	(* Titlezeile zeichnen *)
	FB_TN_SC_FILL(	Iin_X1 := INT#00,
					Iin_Y1 := INT#00,
					Iin_X2 := INT#79,
					Iin_Y2 := INT#00,
					Iby_CHAR := BYTE#32,
					Iby_Attr := BYTE#16#07,
					Xus_TN_SCREEN := Xus_TN_SCREEN);

	(* Fusszeile zeichnen *)
	FB_TN_SC_FILL(	Iin_X1 := INT#00,
					Iin_Y1 := INT#23,
					Iin_X2 := INT#79,
					Iin_Y2 := INT#23,
					Iby_CHAR := BYTE#32,
					Iby_Attr := BYTE#16#37,
					Xus_TN_SCREEN := Xus_TN_SCREEN);

	(* Rahmen für Viewport zeichnen *)
	FB_TN_SC_BOX(	Iin_X1 := INT#00,
					Iin_Y1 := INT#01,
					Iin_X2 := INT#77,
					Iin_Y2 := INT#17,
					Iby_FILL := BYTE#16#00, (* keine Füllung *)
					Iin_BORDER := INT#02, (* Double-Line Border *)
					Iby_ATTR := BYTE#16#74, (* Weiss , Blau *)
					Xus_TN_SCREEN := Xus_TN_SCREEN);

	(* Shadow für Rahmen von Viewport zeichnen *)
	FB_TN_SC_ADD_SHADOW(Iin_X1 := INT#01,
						Iin_Y1 := INT#02,
						Iin_X2 := INT#78,
						Iin_Y2 := INT#18,
						Iin_OPTION := INT#00,
						Xus_TN_SCREEN := Xus_TN_SCREEN);

	(* Trennlinie Viewport_Data und Commandline zeichnen *)
	FB_TN_SC_LINE(	Iin_X1 := INT#00,
					Iin_Y1 := INT#15,
					Iin_X2 := INT#77,
					Iin_Y2 := INT#15,
					Iby_ATTR := BYTE#16#74,
					Iby_BORDER := BYTE#02,
					Xus_TN_SCREEN := Xus_TN_SCREEN);

	(* Title Viewport zeichnen *)
	FB_TN_SC_WRITE(	Iin_X := INT#29,
					Iin_Y := INT#01,
					Iby_ATTR := BYTE#16#74,
					Ist_STRING := '[ SYSTEM-CONSOLE ]',
					Xus_TN_SCREEN := Xus_TN_SCREEN);

	(* Rahmen für Parameter-Feld zeichnen *)
	FB_TN_SC_BOX(	Iin_X1 := INT#02,
					Iin_Y1 := INT#19,
					Iin_X2 := INT#74,
					Iin_Y2 := INT#21,
					Iby_FILL := BYTE#16#20,
					Iin_BORDER := INT#01, (* Double-Line Border *)
					Iby_ATTR := BYTE#16#74, (* Weiss , Blau *)
					Xus_TN_SCREEN := Xus_TN_SCREEN);

	(* Shadow für Rahmen von Parameter-Feld zeichnen *)
	FB_TN_SC_ADD_SHADOW(Iin_X1 := INT#03,
						Iin_Y1 := INT#20,
						Iin_X2 := INT#75,
						Iin_Y2 := INT#22,
						Iin_OPTION := INT#00,
						Xus_TN_SCREEN := Xus_TN_SCREEN);

	(* Alle Input-Controls initialisieren *)

	Xus_TN_INPUT_CONTROL.bo_Enable := FALSE;

	(* Initialisierung der Eingabe-Zeile *)
	Xus_TN_INPUT_CONTROL.usa_TN_INPUT_CONTROL_DATA[1].in_Type := INT#01;
	Xus_TN_INPUT_CONTROL.usa_TN_INPUT_CONTROL_DATA[1].in_Y := INT#16;
	Xus_TN_INPUT_CONTROL.usa_TN_INPUT_CONTROL_DATA[1].in_X := INT#09;
	Xus_TN_INPUT_CONTROL.usa_TN_INPUT_CONTROL_DATA[1].by_Attr_mF := BYTE#16#72; (* Weiss, Grün *)
	Xus_TN_INPUT_CONTROL.usa_TN_INPUT_CONTROL_DATA[1].by_Attr_oF := BYTE#16#74; (* Weiss, Blau *)
	Xus_TN_INPUT_CONTROL.usa_TN_INPUT_CONTROL_DATA[1].in_Cursor_Pos := INT#0;
	Xus_TN_INPUT_CONTROL.usa_TN_INPUT_CONTROL_DATA[1].bo_Input_Only_Num := FALSE;
	Xus_TN_INPUT_CONTROL.usa_TN_INPUT_CONTROL_DATA[1].bo_Input_Hidden := FALSE;
	Xus_TN_INPUT_CONTROL.usa_TN_INPUT_CONTROL_DATA[1].st_Input_Mask := '                                                                    ';
	Xus_TN_INPUT_CONTROL.usa_TN_INPUT_CONTROL_DATA[1].st_Input_Data := Xus_TN_INPUT_CONTROL.usa_TN_INPUT_CONTROL_DATA[1].st_Input_Mask;
	Xus_TN_INPUT_CONTROL.usa_TN_INPUT_CONTROL_DATA[1].st_Input_ToolTip := 'Eingabezeile aktiv       | SCROLL F1/F2/F3/F4 |';
	Xus_TN_INPUT_CONTROL.usa_TN_INPUT_CONTROL_DATA[1].in_Input_Option := INT#02;
	Xus_TN_INPUT_CONTROL.usa_TN_INPUT_CONTROL_DATA[1].in_Title_Y_Offset := INT#00;
	Xus_TN_INPUT_CONTROL.usa_TN_INPUT_CONTROL_DATA[1].in_Title_X_Offset := INT#00;
	Xus_TN_INPUT_CONTROL.usa_TN_INPUT_CONTROL_DATA[1].by_Title_Attr := BYTE#16#34;
	Xus_TN_INPUT_CONTROL.usa_TN_INPUT_CONTROL_DATA[1].st_Title_String := 'Befehl: ';

	(* Initialisierung Selection Text *)
	Xus_TN_INPUT_CONTROL.usa_TN_INPUT_CONTROL_DATA[2].in_Type := INT#03;
	Xus_TN_INPUT_CONTROL.usa_TN_INPUT_CONTROL_DATA[2].in_Y := INT#20;
	Xus_TN_INPUT_CONTROL.usa_TN_INPUT_CONTROL_DATA[2].in_X := INT#18;
	Xus_TN_INPUT_CONTROL.usa_TN_INPUT_CONTROL_DATA[2].by_Attr_mF := BYTE#16#17;
	Xus_TN_INPUT_CONTROL.usa_TN_INPUT_CONTROL_DATA[2].by_Attr_oF := BYTE#16#47;
	Xus_TN_INPUT_CONTROL.usa_TN_INPUT_CONTROL_DATA[2].st_Input_ToolTip := ' aktuellen LOG-Level aendern     | press enter to select |';
	Xus_TN_INPUT_CONTROL.usa_TN_INPUT_CONTROL_DATA[2].in_Input_Option := INT#00;
	Xus_TN_INPUT_CONTROL.usa_TN_INPUT_CONTROL_DATA[2].in_Title_Y_Offset := INT#00;
	Xus_TN_INPUT_CONTROL.usa_TN_INPUT_CONTROL_DATA[2].in_Title_X_Offset := INT#00;
	Xus_TN_INPUT_CONTROL.usa_TN_INPUT_CONTROL_DATA[2].by_Title_Attr := BYTE#16#34;
	Xus_TN_INPUT_CONTROL.usa_TN_INPUT_CONTROL_DATA[2].st_Title_String := ' LOG-Level ';
	Xus_TN_INPUT_CONTROL.usa_TN_INPUT_CONTROL_DATA[2].st_Input_Mask := '  ';
	Xus_TN_INPUT_CONTROL.usa_TN_INPUT_CONTROL_DATA[2].st_Input_Data := '01#02#03#04#05#06#07#08#09#10#11#12#13#14#15';

	(* Initialisierung Selection Text *)
	Xus_TN_INPUT_CONTROL.usa_TN_INPUT_CONTROL_DATA[3].in_Type := INT#02;
	Xus_TN_INPUT_CONTROL.usa_TN_INPUT_CONTROL_DATA[3].in_Y := INT#20;
	Xus_TN_INPUT_CONTROL.usa_TN_INPUT_CONTROL_DATA[3].in_X := INT#37;
	Xus_TN_INPUT_CONTROL.usa_TN_INPUT_CONTROL_DATA[3].by_Attr_mF := BYTE#16#17;
	Xus_TN_INPUT_CONTROL.usa_TN_INPUT_CONTROL_DATA[3].by_Attr_oF := BYTE#16#47;
	Xus_TN_INPUT_CONTROL.usa_TN_INPUT_CONTROL_DATA[3].st_Input_ToolTip := ' Optionline aktiv      | press space to select |';
	Xus_TN_INPUT_CONTROL.usa_TN_INPUT_CONTROL_DATA[3].in_Input_Option := INT#02;
	Xus_TN_INPUT_CONTROL.usa_TN_INPUT_CONTROL_DATA[3].in_Title_Y_Offset := INT#00;
	Xus_TN_INPUT_CONTROL.usa_TN_INPUT_CONTROL_DATA[3].in_Title_X_Offset := INT#00;
	Xus_TN_INPUT_CONTROL.usa_TN_INPUT_CONTROL_DATA[3].by_Title_Attr := BYTE#16#34;
	Xus_TN_INPUT_CONTROL.usa_TN_INPUT_CONTROL_DATA[3].st_Title_String := '  Selektion  ';
	Xus_TN_INPUT_CONTROL.usa_TN_INPUT_CONTROL_DATA[3].st_Input_Mask := '     ';
	Xus_TN_INPUT_CONTROL.usa_TN_INPUT_CONTROL_DATA[3].st_Input_Data := '[ ]#[x]';

	(* Initialisierung Selection Text *)
	Xus_TN_INPUT_CONTROL.usa_TN_INPUT_CONTROL_DATA[4].in_Type := INT#02;
	Xus_TN_INPUT_CONTROL.usa_TN_INPUT_CONTROL_DATA[4].in_Y := INT#20;
	Xus_TN_INPUT_CONTROL.usa_TN_INPUT_CONTROL_DATA[4].in_X := INT#58;
	Xus_TN_INPUT_CONTROL.usa_TN_INPUT_CONTROL_DATA[4].by_Attr_mF := BYTE#16#17;
	Xus_TN_INPUT_CONTROL.usa_TN_INPUT_CONTROL_DATA[4].by_Attr_oF := BYTE#16#47;
	Xus_TN_INPUT_CONTROL.usa_TN_INPUT_CONTROL_DATA[4].st_Input_ToolTip := ' Selektion-Text aktiv      | press space to select |';
	Xus_TN_INPUT_CONTROL.usa_TN_INPUT_CONTROL_DATA[4].in_Input_Option := INT#02;
	Xus_TN_INPUT_CONTROL.usa_TN_INPUT_CONTROL_DATA[4].in_Title_Y_Offset := INT#00;
	Xus_TN_INPUT_CONTROL.usa_TN_INPUT_CONTROL_DATA[4].in_Title_X_Offset := INT#00;
	Xus_TN_INPUT_CONTROL.usa_TN_INPUT_CONTROL_DATA[4].by_Title_Attr := BYTE#16#34;
	Xus_TN_INPUT_CONTROL.usa_TN_INPUT_CONTROL_DATA[4].st_Title_String := ' Betriebsart ';
	Xus_TN_INPUT_CONTROL.usa_TN_INPUT_CONTROL_DATA[4].st_Input_Mask := '               ';
	Xus_TN_INPUT_CONTROL.usa_TN_INPUT_CONTROL_DATA[4].st_Input_Data := '<Auto>#<Hand>#<Einzelschritt>#<Stop>#<Restart>';

	(* Control-Tool-Tip *)
	Xus_TN_INPUT_CONTROL.in_ToolTip_Y := INT#23;
	Xus_TN_INPUT_CONTROL.in_ToolTip_X := INT#00;
	Xus_TN_INPUT_CONTROL.by_ToolTip_Attr := BYTE#16#37;
	Xus_TN_INPUT_CONTROL.in_ToolTip_Size := INT#60;

	(* Control-Verwaltung initialisieren *)
	Xus_TN_INPUT_CONTROL.in_Count := INT#04;
	Xus_TN_INPUT_CONTROL.bo_Enable := TRUE;
	Xus_TN_INPUT_CONTROL.bo_Reset_Fokus := TRUE;

	(* LOG-Viewport initialisieren und Neuzeichnen auslösen *)
	us_LOG_VIEWPORT.COUNT := 13;
	us_LOG_VIEWPORT.UPDATE := TRUE;

	(* Menu initialisieren *)
	Xus_TN_MENU.in_X := INT#00;
	Xus_TN_MENU.in_Y := INT#00;
	Xus_TN_MENU.by_Attr_mF := BYTE#16#33; (* yellow + brown *)
	Xus_TN_MENU.by_Attr_oF := BYTE#16#0F; (* schwarz + grau *)
	Xus_TN_MENU.st_MENU_TEXT := 'Datei#Bearbeiten#Ansicht#Ende';
	Xus_TN_MENU.st_MENU_TEXT := CONCAT(Xus_TN_MENU.st_MENU_TEXT,'%oeffnen#-#speichern#beenden%loeschen#-#einfuegen#-#kopieren');
	Xus_TN_MENU.st_MENU_TEXT := CONCAT(Xus_TN_MENU.st_MENU_TEXT,'%alles#detail#kopieren%Logout');
	Xus_TN_MENU.bo_Create := TRUE;

END_IF;

IF (Xus_TN_SCREEN.in_Page_Number = INT#11) THEN

	(* Eingabezeile: Befehl -> eingegebenen String übernehmen *)
	IF (Xus_TN_INPUT_CONTROL.usa_TN_INPUT_CONTROL_DATA[1].bo_Input_Entered = TRUE) THEN

		Xus_TN_INPUT_CONTROL.usa_TN_INPUT_CONTROL_DATA[1].bo_Input_Entered := FALSE;
		Gst_SysLog_Command := Xus_TN_INPUT_CONTROL.usa_TN_INPUT_CONTROL_DATA[1].st_Input_String;

	END_IF;

	(* Eingabezeile: LOG_LEVEL -> eingegebenen String übernehmen *)
	IF (Xus_TN_INPUT_CONTROL.usa_TN_INPUT_CONTROL_DATA[2].bo_Input_Entered = TRUE) THEN

		Xus_TN_INPUT_CONTROL.usa_TN_INPUT_CONTROL_DATA[2].bo_Input_Entered := FALSE;
		Gst_SysLog_Command := CONCAT('LOG_LEVEL ',Xus_TN_INPUT_CONTROL.usa_TN_INPUT_CONTROL_DATA[2].st_Input_String);

	END_IF;

	(* LOG-Viewport - Scroll Funktionen *)
	IF (Xus_TN_INPUT_CONTROL.in_Focus_at = INT#01) THEN
		CASE BYTE_TO_INT(Xus_TN_SCREEN.by_Input_Exten_Code) OF
		80: (* F1 Taste *)
			us_LOG_VIEWPORT.MOVE_TO_X := 30001; (* Scrollen zum Listenanfang *)
		81: (* F2 Taste *)
			us_LOG_VIEWPORT.MOVE_TO_X := us_LOG_VIEWPORT.COUNT; (* Scrollen eine Seite nach oben *)
		82: (* F3 Taste *)
			us_LOG_VIEWPORT.MOVE_TO_X := 0 - us_LOG_VIEWPORT.COUNT;
		83: (* F4 Taste *)
			us_LOG_VIEWPORT.MOVE_TO_X := 30000; (* Scrollen zum Listenende *)
		END_CASE;
	END_IF;

	(* LOG-Viewport Updaten *)
	FB_LOG_VIEWPORT(LC := LOG_CL,
					LV := us_LOG_VIEWPORT);

	(* LOG-Viewport zeichnen *)
	FB_TN_SC_VIEWPORT(	Xus_LOG_VIEWPORT := us_LOG_VIEWPORT,
						Xus_LOG_CONTROL := LOG_CL,
						Xus_TN_SCREEN := Xus_TN_SCREEN,
						Iin_X := INT#01,
						Iin_Y := INT#02,
						Iin_Width := INT#76,
						Idw_ATTR_1 := DWORD#16#64542434, (* Color + Level 3:2:1:0 *)
						Idw_ATTR_2 := DWORD#16#94047414, (* Color + Level 7:6:5:4 *)
						Iti_TIME := TIME#100ms);
END_IF;

IF LEN(Gst_SysLog_Command) > 0 THEN

	(* Kommando echo *)
	LOG_CL.NEW_MSG := CONCAT('ACTION: ',Gst_SysLog_Command);
	LOG_CL.NEW_MSG_OPTION := 0;
	FB_LOG_MESSAGE();

	Gst_SysLog_Command := '';

END_IF;

END_PROGRAM

// POUs/DEMO/TN_VISION_DEMO_2
PROGRAM TN_VISION_DEMO_2
VAR
	FB_TN_FRAMEWORK : TN_FRAMEWORK;
	FB_TN_SC_FILL : TN_SC_FILL;
	FB_TN_SC_WRITE_C : TN_SC_WRITE_C;
	FB_TN_SC_WRITE : TN_SC_WRITE;
	Xus_TN_MENU : us_TN_MENU;
	Xus_TN_INPUT_CONTROL : us_TN_INPUT_CONTROL;
	Xus_TN_SCREEN : us_TN_SCREEN;
	S_BUF : NETWORK_BUFFER;
	R_BUF : NETWORK_BUFFER;
	IP_C : IP_C;
END_VAR

FB_TN_FRAMEWORK(
					us_TN_INPUT_CONTROL := Xus_TN_INPUT_CONTROL ,
					us_TN_SCREEN := Xus_TN_SCREEN ,
					us_TN_MENU := Xus_TN_MENU ,
					S_BUF := S_BUF ,
					R_BUF:= R_BUF ,
					IP_C:= IP_C ,
					PORT := WORD#0
					 );


(* Initialisierung der Daten und Strukturen *)
IF (Xus_TN_SCREEN.in_Page_Number = INT#00) THEN
	Xus_TN_SCREEN.in_Page_Number := INT#01;

	(* Clear-Screen (Farbe setzen + Display löschen) *)
	Xus_TN_SCREEN.by_Clear_Screen_Attr := BYTE#16#00;
	Xus_TN_SCREEN.bo_Clear_Screen := TRUE;

	(* Screen initialisieren (mit Leerzeichen füllen) *)
	FB_TN_SC_FILL(	Iin_X1 := INT#00,
					Iin_Y1 := INT#00,
					Iin_X2 := INT#79,
					Iin_Y2 := INT#23,
					Iby_CHAR := BYTE#32,
					Iby_Attr := BYTE#16#00,
					Xus_TN_SCREEN := Xus_TN_SCREEN);

	(* Statische Texte ausgeben *)
	FB_TN_SC_WRITE(	Iin_X := INT#00,
					Iin_Y := INT#00,
					Iby_ATTR := BYTE#16#70,
					Ist_STRING := 'Login Screen                                                     FL SWITCH MM HS',
					Xus_TN_SCREEN := Xus_TN_SCREEN);

	(* Statische Texte ausgeben *)
	FB_TN_SC_WRITE(	Iin_X := INT#00,
					Iin_Y := INT#03,
					Iby_ATTR := BYTE#16#70,
					Ist_STRING := 'XXXXXXXXX',
					Xus_TN_SCREEN := Xus_TN_SCREEN);

	(* Statische Texte ausgeben *)
	FB_TN_SC_WRITE(	Iin_X := INT#00,
					Iin_Y := INT#04,
					Iby_ATTR := BYTE#16#70,
					Ist_STRING := 'X   X  XX',
					Xus_TN_SCREEN := Xus_TN_SCREEN);

	(* Statische Texte ausgeben *)
	FB_TN_SC_WRITE(	Iin_X := INT#00,
					Iin_Y := INT#05,
					Iby_ATTR := BYTE#16#70,
					Ist_STRING := 'X   O   X      ---> Phoenix Contact Managed Switch System <---',
					Xus_TN_SCREEN := Xus_TN_SCREEN);

	(* Statische Texte ausgeben *)
	FB_TN_SC_WRITE(	Iin_X := INT#00,
					Iin_Y := INT#06,
					Iby_ATTR := BYTE#16#70,
					Ist_STRING := 'X   X  XX               Phoenix Contact GmbH & Co KG',
					Xus_TN_SCREEN := Xus_TN_SCREEN);

	(* Statische Texte ausgeben *)
	FB_TN_SC_WRITE(	Iin_X := INT#00,
					Iin_Y := INT#07,
					Iby_ATTR := BYTE#16#70,
					Ist_STRING := 'X   XXXXX                   www.PhoenixContact.com',
					Xus_TN_SCREEN := Xus_TN_SCREEN);

	(* Statische Texte ausgeben *)
	FB_TN_SC_WRITE(	Iin_X := INT#00,
					Iin_Y := INT#08,
					Iby_ATTR := BYTE#16#70,
					Ist_STRING := 'X   XXXXX',
					Xus_TN_SCREEN := Xus_TN_SCREEN);

	(* Statische Texte ausgeben *)
	FB_TN_SC_WRITE(	Iin_X := INT#00,
					Iin_Y := INT#09,
					Iby_ATTR := BYTE#16#70,
					Ist_STRING := 'XXXXXXXXX',
					Xus_TN_SCREEN := Xus_TN_SCREEN);

	(* Statische Texte ausgeben *)
	FB_TN_SC_WRITE(	Iin_X := INT#00,
					Iin_Y := INT#11,
					Iby_ATTR := BYTE#16#70,
					Ist_STRING := '                Running switch application version:  4.00',
					Xus_TN_SCREEN := Xus_TN_SCREEN);

	(* Alle Input-Controls initialisieren *)

	Xus_TN_INPUT_CONTROL.bo_Enable := FALSE;

  (* Initialisierung der Eingabe-Zeile *)
	Xus_TN_INPUT_CONTROL.usa_TN_INPUT_CONTROL_DATA[1].in_Type := INT#01;
	Xus_TN_INPUT_CONTROL.usa_TN_INPUT_CONTROL_DATA[1].in_Y := INT#17;
	Xus_TN_INPUT_CONTROL.usa_TN_INPUT_CONTROL_DATA[1].in_X := INT#33;
	Xus_TN_INPUT_CONTROL.usa_TN_INPUT_CONTROL_DATA[1].by_Attr_mF := BYTE#16#70;
	Xus_TN_INPUT_CONTROL.usa_TN_INPUT_CONTROL_DATA[1].by_Attr_oF := BYTE#16#70;
	Xus_TN_INPUT_CONTROL.usa_TN_INPUT_CONTROL_DATA[1].in_Cursor_Pos := INT#0;
	Xus_TN_INPUT_CONTROL.usa_TN_INPUT_CONTROL_DATA[1].bo_Input_Only_Num := FALSE;
	Xus_TN_INPUT_CONTROL.usa_TN_INPUT_CONTROL_DATA[1].bo_Input_Hidden := TRUE;
	Xus_TN_INPUT_CONTROL.usa_TN_INPUT_CONTROL_DATA[1].st_Input_Mask := '                ';
	Xus_TN_INPUT_CONTROL.usa_TN_INPUT_CONTROL_DATA[1].st_Input_Data := Xus_TN_INPUT_CONTROL.usa_TN_INPUT_CONTROL_DATA[1].st_Input_Mask;
	Xus_TN_INPUT_CONTROL.usa_TN_INPUT_CONTROL_DATA[1].st_Input_ToolTip := '';
	Xus_TN_INPUT_CONTROL.usa_TN_INPUT_CONTROL_DATA[1].in_Input_Option := INT#00;
	Xus_TN_INPUT_CONTROL.usa_TN_INPUT_CONTROL_DATA[1].in_Title_Y_Offset := INT#00;
	Xus_TN_INPUT_CONTROL.usa_TN_INPUT_CONTROL_DATA[1].in_Title_X_Offset := -12;
	Xus_TN_INPUT_CONTROL.usa_TN_INPUT_CONTROL_DATA[1].by_Title_Attr := BYTE#16#70;
	Xus_TN_INPUT_CONTROL.usa_TN_INPUT_CONTROL_DATA[1].st_Title_String := 'Password:  [                ]';

	(* Control-Tool-Tip *)
	Xus_TN_INPUT_CONTROL.in_ToolTip_Y := INT#23;
	Xus_TN_INPUT_CONTROL.in_ToolTip_X := INT#09;
	Xus_TN_INPUT_CONTROL.by_ToolTip_Attr := BYTE#16#70;
	Xus_TN_INPUT_CONTROL.in_ToolTip_Size := INT#30;

	(* Control-Verwaltung initialisieren *)
	Xus_TN_INPUT_CONTROL.in_Count := INT#01;
	Xus_TN_INPUT_CONTROL.bo_Enable := TRUE;
	Xus_TN_INPUT_CONTROL.bo_Reset_Fokus := TRUE;
END_IF;

IF (Xus_TN_SCREEN.in_Page_Number = INT#01) THEN

	(* eingegebenen String übernehmen *)
	IF Xus_TN_INPUT_CONTROL.usa_TN_INPUT_CONTROL_DATA[1].bo_Input_Entered = TRUE THEN

		Xus_TN_INPUT_CONTROL.usa_TN_INPUT_CONTROL_DATA[1].bo_Input_Entered := FALSE;

		Xus_TN_INPUT_CONTROL.usa_TN_INPUT_CONTROL_DATA[1].st_Input_String :=
			OSCAT_BASIC.LOWERCASE(str:=Xus_TN_INPUT_CONTROL.usa_TN_INPUT_CONTROL_DATA[1].st_Input_String);

		IF Xus_TN_INPUT_CONTROL.usa_TN_INPUT_CONTROL_DATA[1].st_Input_String = 'oscat' THEN
			Xus_TN_SCREEN.in_Page_Number := INT#04;

		ELSE
			FB_TN_SC_WRITE_C(	Iin_Y := Xus_TN_INPUT_CONTROL.in_ToolTip_Y,
								Iin_X := Xus_TN_INPUT_CONTROL.in_ToolTip_X,
								Iby_ATTR := BYTE#16#F1,
								Iin_OPTION := INT#02, (* Center-String *)
								Iin_LENGTH := Xus_TN_INPUT_CONTROL.in_ToolTip_Size,
								Ist_STRING := ' User Password Failed   ',
								Xus_TN_SCREEN := Xus_TN_SCREEN);
		END_IF;
	END_IF;
END_IF;

(* Initialisierung der Daten und Strukturen *)
IF (Xus_TN_SCREEN.in_Page_Number = INT#04) THEN
	Xus_TN_SCREEN.in_Page_Number := INT#05;

	(* Clear-Screen (Farbe setzen + Display löschen) *)
	Xus_TN_SCREEN.by_Clear_Screen_Attr := BYTE#16#00;
	Xus_TN_SCREEN.bo_Clear_Screen := TRUE;

	(* Screen initialisieren (mit Leerzeichen füllen) *)
	FB_TN_SC_FILL(	Iin_X1 := INT#00,
					Iin_Y1 := INT#00,
					Iin_X2 := INT#79,
					Iin_Y2 := INT#23,
					Iby_CHAR := BYTE#32,
					Iby_Attr := BYTE#16#00,
					Xus_TN_SCREEN := Xus_TN_SCREEN);

	(* Statische Texte ausgeben *)
	FB_TN_SC_WRITE(	Iin_X := INT#00,
					Iin_Y := INT#00,
					Iby_ATTR := BYTE#16#70,
					Ist_STRING := 'Basic Switch Configuration                                       FL SWITCH MM HS',
					Xus_TN_SCREEN := Xus_TN_SCREEN);

	(* Statische Texte ausgeben                                         *)
	FB_TN_SC_WRITE(	Iin_X := INT#00,
					Iin_Y := INT#03,
					Iby_ATTR := BYTE#16#70,
					Ist_STRING := 'XXXXXXXXX        MAC Address             : 00:A0:45:00:6E:9B',
					Xus_TN_SCREEN := Xus_TN_SCREEN);

	(* Statische Texte ausgeben *)
	FB_TN_SC_WRITE(	Iin_X := INT#00,
					Iin_Y := INT#04,
					Iby_ATTR := BYTE#16#70,
					Ist_STRING := 'X   X  XX',
					Xus_TN_SCREEN := Xus_TN_SCREEN);

	(* Statische Texte ausgeben *)
	FB_TN_SC_WRITE(	Iin_X := INT#00,
					Iin_Y := INT#05,
					Iby_ATTR := BYTE#16#70,
					Ist_STRING := 'X   O   X',
					Xus_TN_SCREEN := Xus_TN_SCREEN);

	(* Statische Texte ausgeben *)
	FB_TN_SC_WRITE(	Iin_X := INT#00,
					Iin_Y := INT#06,
					Iby_ATTR := BYTE#16#70,
					Ist_STRING := 'X   X  XX',
					Xus_TN_SCREEN := Xus_TN_SCREEN);

	(* Statische Texte ausgeben *)
	FB_TN_SC_WRITE(	Iin_X := INT#00,
					Iin_Y := INT#07,
					Iby_ATTR := BYTE#16#70,
					Ist_STRING := 'X   XXXXX',
					Xus_TN_SCREEN := Xus_TN_SCREEN);

	(* Statische Texte ausgeben *)
	FB_TN_SC_WRITE(	Iin_X := INT#00,
					Iin_Y := INT#08,
					Iby_ATTR := BYTE#16#70,
					Ist_STRING := 'X   XXXXX',
					Xus_TN_SCREEN := Xus_TN_SCREEN);

	(* Statische Texte ausgeben *)
	FB_TN_SC_WRITE(	Iin_X := INT#00,
					Iin_Y := INT#09,
					Iby_ATTR := BYTE#16#70,
					Ist_STRING := 'XXXXXXXXX',
					Xus_TN_SCREEN := Xus_TN_SCREEN);

	(* Alle Input-Controls initialisieren *)

	Xus_TN_INPUT_CONTROL.bo_Enable      := FALSE;

	Xus_TN_INPUT_CONTROL.usa_TN_INPUT_CONTROL_DATA[1].in_Type := INT#01;
	Xus_TN_INPUT_CONTROL.usa_TN_INPUT_CONTROL_DATA[1].in_Y := INT#04;
	Xus_TN_INPUT_CONTROL.usa_TN_INPUT_CONTROL_DATA[1].in_X := INT#44;
	Xus_TN_INPUT_CONTROL.usa_TN_INPUT_CONTROL_DATA[1].by_Attr_mF := BYTE#16#07; (* Weiss, Grün *)
	Xus_TN_INPUT_CONTROL.usa_TN_INPUT_CONTROL_DATA[1].by_Attr_oF := BYTE#16#70; (* Weiss, Blau *)
	Xus_TN_INPUT_CONTROL.usa_TN_INPUT_CONTROL_DATA[1].in_Cursor_Pos := INT#0;
	Xus_TN_INPUT_CONTROL.usa_TN_INPUT_CONTROL_DATA[1].bo_Input_Only_Num := TRUE;
	Xus_TN_INPUT_CONTROL.usa_TN_INPUT_CONTROL_DATA[1].bo_Input_Hidden := FALSE;
	Xus_TN_INPUT_CONTROL.usa_TN_INPUT_CONTROL_DATA[1].st_Input_Mask := '   .   .   .   ';
	Xus_TN_INPUT_CONTROL.usa_TN_INPUT_CONTROL_DATA[1].st_Input_Data := Xus_TN_INPUT_CONTROL.usa_TN_INPUT_CONTROL_DATA[1].st_Input_Mask;
	Xus_TN_INPUT_CONTROL.usa_TN_INPUT_CONTROL_DATA[1].st_Input_ToolTip := 'Enter Agent IP Address in decimal dot format (e.g., 209.131.209.13)';
	Xus_TN_INPUT_CONTROL.usa_TN_INPUT_CONTROL_DATA[1].in_Input_Option := INT#01;
	Xus_TN_INPUT_CONTROL.usa_TN_INPUT_CONTROL_DATA[1].in_Title_Y_Offset := INT#00;
	Xus_TN_INPUT_CONTROL.usa_TN_INPUT_CONTROL_DATA[1].in_Title_X_Offset := -27;
	Xus_TN_INPUT_CONTROL.usa_TN_INPUT_CONTROL_DATA[1].by_Title_Attr := BYTE#16#70;
	Xus_TN_INPUT_CONTROL.usa_TN_INPUT_CONTROL_DATA[1].st_Title_String := 'IP Address              : [149.208.100.100]';

	Xus_TN_INPUT_CONTROL.usa_TN_INPUT_CONTROL_DATA[2].in_Type := INT#01;
	Xus_TN_INPUT_CONTROL.usa_TN_INPUT_CONTROL_DATA[2].in_Y := INT#05;
	Xus_TN_INPUT_CONTROL.usa_TN_INPUT_CONTROL_DATA[2].in_X := INT#44;
	Xus_TN_INPUT_CONTROL.usa_TN_INPUT_CONTROL_DATA[2].by_Attr_mF := BYTE#16#07; (* Weiss, Grün *)
	Xus_TN_INPUT_CONTROL.usa_TN_INPUT_CONTROL_DATA[2].by_Attr_oF := BYTE#16#70; (* Weiss, Blau *)
	Xus_TN_INPUT_CONTROL.usa_TN_INPUT_CONTROL_DATA[2].in_Cursor_Pos := INT#0;
	Xus_TN_INPUT_CONTROL.usa_TN_INPUT_CONTROL_DATA[2].bo_Input_Only_Num := TRUE;
	Xus_TN_INPUT_CONTROL.usa_TN_INPUT_CONTROL_DATA[2].bo_Input_Hidden := FALSE;
	Xus_TN_INPUT_CONTROL.usa_TN_INPUT_CONTROL_DATA[2].st_Input_Mask := '   .   .   .   ';
	Xus_TN_INPUT_CONTROL.usa_TN_INPUT_CONTROL_DATA[2].st_Input_Data := Xus_TN_INPUT_CONTROL.usa_TN_INPUT_CONTROL_DATA[1].st_Input_Mask;
	Xus_TN_INPUT_CONTROL.usa_TN_INPUT_CONTROL_DATA[2].st_Input_ToolTip := 'Enter Agent Netmask (e.g., 255.255.255.0)';
	Xus_TN_INPUT_CONTROL.usa_TN_INPUT_CONTROL_DATA[2].in_Input_Option := INT#01;
	Xus_TN_INPUT_CONTROL.usa_TN_INPUT_CONTROL_DATA[2].in_Title_Y_Offset := INT#00;
	Xus_TN_INPUT_CONTROL.usa_TN_INPUT_CONTROL_DATA[2].in_Title_X_Offset := -27;
	Xus_TN_INPUT_CONTROL.usa_TN_INPUT_CONTROL_DATA[2].by_Title_Attr := BYTE#16#70;
	Xus_TN_INPUT_CONTROL.usa_TN_INPUT_CONTROL_DATA[2].st_Title_String := 'Subnet Mask             : [255.255.255.128]';

	Xus_TN_INPUT_CONTROL.usa_TN_INPUT_CONTROL_DATA[3].in_Type := INT#01;
	Xus_TN_INPUT_CONTROL.usa_TN_INPUT_CONTROL_DATA[3].in_Y := INT#06;
	Xus_TN_INPUT_CONTROL.usa_TN_INPUT_CONTROL_DATA[3].in_X := INT#44;
	Xus_TN_INPUT_CONTROL.usa_TN_INPUT_CONTROL_DATA[3].by_Attr_mF := BYTE#16#07; (* Weiss, Grün *)
	Xus_TN_INPUT_CONTROL.usa_TN_INPUT_CONTROL_DATA[3].by_Attr_oF := BYTE#16#70; (* Weiss, Blau *)
	Xus_TN_INPUT_CONTROL.usa_TN_INPUT_CONTROL_DATA[3].in_Cursor_Pos := INT#0;
	Xus_TN_INPUT_CONTROL.usa_TN_INPUT_CONTROL_DATA[3].bo_Input_Only_Num := TRUE;
	Xus_TN_INPUT_CONTROL.usa_TN_INPUT_CONTROL_DATA[3].bo_Input_Hidden := FALSE;
	Xus_TN_INPUT_CONTROL.usa_TN_INPUT_CONTROL_DATA[3].st_Input_Mask := '   .   .   .   ';
	Xus_TN_INPUT_CONTROL.usa_TN_INPUT_CONTROL_DATA[3].st_Input_Data := Xus_TN_INPUT_CONTROL.usa_TN_INPUT_CONTROL_DATA[1].st_Input_Mask;
	Xus_TN_INPUT_CONTROL.usa_TN_INPUT_CONTROL_DATA[3].st_Input_ToolTip := 'Enter Agent Default Gateway, (e.g., 209.131.209.1)';
	Xus_TN_INPUT_CONTROL.usa_TN_INPUT_CONTROL_DATA[3].in_Input_Option := INT#01;
	Xus_TN_INPUT_CONTROL.usa_TN_INPUT_CONTROL_DATA[3].in_Title_Y_Offset := INT#00;
	Xus_TN_INPUT_CONTROL.usa_TN_INPUT_CONTROL_DATA[3].in_Title_X_Offset := -27;
	Xus_TN_INPUT_CONTROL.usa_TN_INPUT_CONTROL_DATA[3].by_Title_Attr := BYTE#16#70;
	Xus_TN_INPUT_CONTROL.usa_TN_INPUT_CONTROL_DATA[3].st_Title_String := 'Default Gateway         : [149.208.100.1  ]';

	Xus_TN_INPUT_CONTROL.usa_TN_INPUT_CONTROL_DATA[4].in_Type := INT#02;
	Xus_TN_INPUT_CONTROL.usa_TN_INPUT_CONTROL_DATA[4].in_Y := INT#07;
	Xus_TN_INPUT_CONTROL.usa_TN_INPUT_CONTROL_DATA[4].in_X := INT#44;
	Xus_TN_INPUT_CONTROL.usa_TN_INPUT_CONTROL_DATA[4].by_Attr_mF := BYTE#16#07;
	Xus_TN_INPUT_CONTROL.usa_TN_INPUT_CONTROL_DATA[4].by_Attr_oF := BYTE#16#70;
	Xus_TN_INPUT_CONTROL.usa_TN_INPUT_CONTROL_DATA[4].st_Input_Mask := '       ';
	Xus_TN_INPUT_CONTROL.usa_TN_INPUT_CONTROL_DATA[4].st_Input_Data := 'BootP  #DHCP   #DCP    #Static ';
	Xus_TN_INPUT_CONTROL.usa_TN_INPUT_CONTROL_DATA[4].st_Input_ToolTip := 'Push SPACE to select the address assignment (effective after reboot)';
	Xus_TN_INPUT_CONTROL.usa_TN_INPUT_CONTROL_DATA[4].in_Input_Option := INT#02;
	Xus_TN_INPUT_CONTROL.usa_TN_INPUT_CONTROL_DATA[4].in_Title_Y_Offset := INT#00;
	Xus_TN_INPUT_CONTROL.usa_TN_INPUT_CONTROL_DATA[4].in_Title_X_Offset := -27;
	Xus_TN_INPUT_CONTROL.usa_TN_INPUT_CONTROL_DATA[4].by_Title_Attr := BYTE#16#70;
	Xus_TN_INPUT_CONTROL.usa_TN_INPUT_CONTROL_DATA[4].st_Title_String := 'IP Parameter Assignment : <BootP  >';

	Xus_TN_INPUT_CONTROL.usa_TN_INPUT_CONTROL_DATA[5].in_Type := INT#02;
	Xus_TN_INPUT_CONTROL.usa_TN_INPUT_CONTROL_DATA[5].in_Y := INT#09;
	Xus_TN_INPUT_CONTROL.usa_TN_INPUT_CONTROL_DATA[5].in_X := INT#44;
	Xus_TN_INPUT_CONTROL.usa_TN_INPUT_CONTROL_DATA[5].by_Attr_mF := BYTE#16#07;
	Xus_TN_INPUT_CONTROL.usa_TN_INPUT_CONTROL_DATA[5].by_Attr_oF := BYTE#16#70;
	Xus_TN_INPUT_CONTROL.usa_TN_INPUT_CONTROL_DATA[5].st_Input_Mask := '                              ';
	Xus_TN_INPUT_CONTROL.usa_TN_INPUT_CONTROL_DATA[5].st_Input_Data := 'No Redundancy#Rapid Spanning Tree, Disabled#Rapid Spanning Tree, Enabled';
	Xus_TN_INPUT_CONTROL.usa_TN_INPUT_CONTROL_DATA[5].st_Input_ToolTip := 'Push SPACE to chose redundancy (network disruption for few seconds if enabled)';
	Xus_TN_INPUT_CONTROL.usa_TN_INPUT_CONTROL_DATA[5].in_Input_Option := INT#02;
	Xus_TN_INPUT_CONTROL.usa_TN_INPUT_CONTROL_DATA[5].in_Title_Y_Offset := INT#00;
	Xus_TN_INPUT_CONTROL.usa_TN_INPUT_CONTROL_DATA[5].in_Title_X_Offset := -27;
	Xus_TN_INPUT_CONTROL.usa_TN_INPUT_CONTROL_DATA[5].by_Title_Attr := BYTE#16#70;
	Xus_TN_INPUT_CONTROL.usa_TN_INPUT_CONTROL_DATA[5].st_Title_String := 'Redundancy              : <No Redundancy                 >';

	(* Statische Texte ausgeben *)
	FB_TN_SC_WRITE(	Iin_X := INT#17,
					Iin_Y := INT#10,
					Iby_ATTR := BYTE#16#70,
					Ist_STRING := 'Current Vlan Status     :  VLAN Transparent',
					Xus_TN_SCREEN := Xus_TN_SCREEN);

	Xus_TN_INPUT_CONTROL.usa_TN_INPUT_CONTROL_DATA[6].in_Type := INT#02;
	Xus_TN_INPUT_CONTROL.usa_TN_INPUT_CONTROL_DATA[6].in_Y := INT#11;
	Xus_TN_INPUT_CONTROL.usa_TN_INPUT_CONTROL_DATA[6].in_X := INT#44;
	Xus_TN_INPUT_CONTROL.usa_TN_INPUT_CONTROL_DATA[6].by_Attr_mF := BYTE#16#07;
	Xus_TN_INPUT_CONTROL.usa_TN_INPUT_CONTROL_DATA[6].by_Attr_oF := BYTE#16#70;
	Xus_TN_INPUT_CONTROL.usa_TN_INPUT_CONTROL_DATA[6].st_Input_Mask := '                        ';
	Xus_TN_INPUT_CONTROL.usa_TN_INPUT_CONTROL_DATA[6].st_Input_Data := 'VLAN Transparent#VLAN Tagging';
	Xus_TN_INPUT_CONTROL.usa_TN_INPUT_CONTROL_DATA[6].st_Input_ToolTip := 'Push SPACE to toggle the VLAN Mode (effective after reboot)';
	Xus_TN_INPUT_CONTROL.usa_TN_INPUT_CONTROL_DATA[6].in_Input_Option := INT#02;
	Xus_TN_INPUT_CONTROL.usa_TN_INPUT_CONTROL_DATA[6].in_Title_Y_Offset := INT#00;
	Xus_TN_INPUT_CONTROL.usa_TN_INPUT_CONTROL_DATA[6].in_Title_X_Offset := -27;
	Xus_TN_INPUT_CONTROL.usa_TN_INPUT_CONTROL_DATA[6].by_Title_Attr := BYTE#16#70;
	Xus_TN_INPUT_CONTROL.usa_TN_INPUT_CONTROL_DATA[6].st_Title_String := 'Vlan Mode               : <VLAN Transparent        >';

	Xus_TN_INPUT_CONTROL.usa_TN_INPUT_CONTROL_DATA[7].in_Type := INT#02;
	Xus_TN_INPUT_CONTROL.usa_TN_INPUT_CONTROL_DATA[7].in_Y := INT#12;
	Xus_TN_INPUT_CONTROL.usa_TN_INPUT_CONTROL_DATA[7].in_X := INT#44;
	Xus_TN_INPUT_CONTROL.usa_TN_INPUT_CONTROL_DATA[7].by_Attr_mF := BYTE#16#07;
	Xus_TN_INPUT_CONTROL.usa_TN_INPUT_CONTROL_DATA[7].by_Attr_oF := BYTE#16#70;
	Xus_TN_INPUT_CONTROL.usa_TN_INPUT_CONTROL_DATA[7].st_Input_Mask := '       ';
	Xus_TN_INPUT_CONTROL.usa_TN_INPUT_CONTROL_DATA[7].st_Input_Data := 'Disable#Enable';
	Xus_TN_INPUT_CONTROL.usa_TN_INPUT_CONTROL_DATA[7].st_Input_ToolTip := 'Push SPACE to Enable/Disable Port Security';
	Xus_TN_INPUT_CONTROL.usa_TN_INPUT_CONTROL_DATA[7].in_Input_Option := INT#02;
	Xus_TN_INPUT_CONTROL.usa_TN_INPUT_CONTROL_DATA[7].in_Title_Y_Offset := INT#00;
	Xus_TN_INPUT_CONTROL.usa_TN_INPUT_CONTROL_DATA[7].in_Title_X_Offset := -27;
	Xus_TN_INPUT_CONTROL.usa_TN_INPUT_CONTROL_DATA[7].by_Title_Attr := BYTE#16#70;
	Xus_TN_INPUT_CONTROL.usa_TN_INPUT_CONTROL_DATA[7].st_Title_String := 'Port Security           : <Disable>';

	Xus_TN_INPUT_CONTROL.usa_TN_INPUT_CONTROL_DATA[8].in_Type := INT#02;
	Xus_TN_INPUT_CONTROL.usa_TN_INPUT_CONTROL_DATA[8].in_Y := INT#13;
	Xus_TN_INPUT_CONTROL.usa_TN_INPUT_CONTROL_DATA[8].in_X := INT#44;
	Xus_TN_INPUT_CONTROL.usa_TN_INPUT_CONTROL_DATA[8].by_Attr_mF := BYTE#16#07;
	Xus_TN_INPUT_CONTROL.usa_TN_INPUT_CONTROL_DATA[8].by_Attr_oF := BYTE#16#70;
	Xus_TN_INPUT_CONTROL.usa_TN_INPUT_CONTROL_DATA[8].st_Input_Mask := '       ';
	Xus_TN_INPUT_CONTROL.usa_TN_INPUT_CONTROL_DATA[8].st_Input_Data := 'Disable#Enable';
	Xus_TN_INPUT_CONTROL.usa_TN_INPUT_CONTROL_DATA[8].st_Input_ToolTip := 'Push SPACE to Enable/Disable Access Control for the WEB Interface';
	Xus_TN_INPUT_CONTROL.usa_TN_INPUT_CONTROL_DATA[8].in_Input_Option := INT#02;
	Xus_TN_INPUT_CONTROL.usa_TN_INPUT_CONTROL_DATA[8].in_Title_Y_Offset := INT#00;
	Xus_TN_INPUT_CONTROL.usa_TN_INPUT_CONTROL_DATA[8].in_Title_X_Offset := -27;
	Xus_TN_INPUT_CONTROL.usa_TN_INPUT_CONTROL_DATA[8].by_Title_Attr := BYTE#16#70;
	Xus_TN_INPUT_CONTROL.usa_TN_INPUT_CONTROL_DATA[8].st_Title_String := 'Access Control for Web  : <Disable>';

	Xus_TN_INPUT_CONTROL.usa_TN_INPUT_CONTROL_DATA[9].in_Type := INT#02;
	Xus_TN_INPUT_CONTROL.usa_TN_INPUT_CONTROL_DATA[9].in_Y := INT#14;
	Xus_TN_INPUT_CONTROL.usa_TN_INPUT_CONTROL_DATA[9].in_X := INT#44;
	Xus_TN_INPUT_CONTROL.usa_TN_INPUT_CONTROL_DATA[9].by_Attr_mF := BYTE#16#07;
	Xus_TN_INPUT_CONTROL.usa_TN_INPUT_CONTROL_DATA[9].by_Attr_oF := BYTE#16#70;
	Xus_TN_INPUT_CONTROL.usa_TN_INPUT_CONTROL_DATA[9].st_Input_Mask := '        ';
	Xus_TN_INPUT_CONTROL.usa_TN_INPUT_CONTROL_DATA[9].st_Input_Data := 'Default#Profinet';
	Xus_TN_INPUT_CONTROL.usa_TN_INPUT_CONTROL_DATA[9].st_Input_ToolTip := 'Push SPACE to select the switch operating mode';
	Xus_TN_INPUT_CONTROL.usa_TN_INPUT_CONTROL_DATA[9].in_Input_Option := INT#02;
	Xus_TN_INPUT_CONTROL.usa_TN_INPUT_CONTROL_DATA[9].in_Title_Y_Offset := INT#00;
	Xus_TN_INPUT_CONTROL.usa_TN_INPUT_CONTROL_DATA[9].in_Title_X_Offset := -27;
	Xus_TN_INPUT_CONTROL.usa_TN_INPUT_CONTROL_DATA[9].by_Title_Attr := BYTE#16#70;
	Xus_TN_INPUT_CONTROL.usa_TN_INPUT_CONTROL_DATA[9].st_Title_String := 'Switch Operating Mode   : <Default >';

	Xus_TN_INPUT_CONTROL.usa_TN_INPUT_CONTROL_DATA[10].in_Type := INT#02;
	Xus_TN_INPUT_CONTROL.usa_TN_INPUT_CONTROL_DATA[10].in_Y := INT#16;
	Xus_TN_INPUT_CONTROL.usa_TN_INPUT_CONTROL_DATA[10].in_X := INT#44;
	Xus_TN_INPUT_CONTROL.usa_TN_INPUT_CONTROL_DATA[10].by_Attr_mF := BYTE#16#07;
	Xus_TN_INPUT_CONTROL.usa_TN_INPUT_CONTROL_DATA[10].by_Attr_oF := BYTE#16#70;
	Xus_TN_INPUT_CONTROL.usa_TN_INPUT_CONTROL_DATA[10].st_Input_Mask := '       ';
	Xus_TN_INPUT_CONTROL.usa_TN_INPUT_CONTROL_DATA[10].st_Input_Data := 'Enable#Disable';
	Xus_TN_INPUT_CONTROL.usa_TN_INPUT_CONTROL_DATA[10].st_Input_ToolTip := 'Push SPACE to Enable/Disable Web Interface (effective after reboot)';
	Xus_TN_INPUT_CONTROL.usa_TN_INPUT_CONTROL_DATA[10].in_Input_Option := INT#02;
	Xus_TN_INPUT_CONTROL.usa_TN_INPUT_CONTROL_DATA[10].in_Title_Y_Offset := INT#00;
	Xus_TN_INPUT_CONTROL.usa_TN_INPUT_CONTROL_DATA[10].in_Title_X_Offset := -27;
	Xus_TN_INPUT_CONTROL.usa_TN_INPUT_CONTROL_DATA[10].by_Title_Attr := BYTE#16#70;
	Xus_TN_INPUT_CONTROL.usa_TN_INPUT_CONTROL_DATA[10].st_Title_String := 'Web Interface           : <Enable >';

	Xus_TN_INPUT_CONTROL.usa_TN_INPUT_CONTROL_DATA[11].in_Type := INT#02;
	Xus_TN_INPUT_CONTROL.usa_TN_INPUT_CONTROL_DATA[11].in_Y := INT#17;
	Xus_TN_INPUT_CONTROL.usa_TN_INPUT_CONTROL_DATA[11].in_X := INT#44;
	Xus_TN_INPUT_CONTROL.usa_TN_INPUT_CONTROL_DATA[11].by_Attr_mF := BYTE#16#07;
	Xus_TN_INPUT_CONTROL.usa_TN_INPUT_CONTROL_DATA[11].by_Attr_oF := BYTE#16#70;
	Xus_TN_INPUT_CONTROL.usa_TN_INPUT_CONTROL_DATA[11].st_Input_Mask := '       ';
	Xus_TN_INPUT_CONTROL.usa_TN_INPUT_CONTROL_DATA[11].st_Input_Data := 'Enable#Disable';
	Xus_TN_INPUT_CONTROL.usa_TN_INPUT_CONTROL_DATA[11].st_Input_ToolTip := 'Push SPACE to Enable/Disable Telnet Interface (effective after reboot)';
	Xus_TN_INPUT_CONTROL.usa_TN_INPUT_CONTROL_DATA[11].in_Input_Option := INT#02;
	Xus_TN_INPUT_CONTROL.usa_TN_INPUT_CONTROL_DATA[11].in_Title_Y_Offset := INT#00;
	Xus_TN_INPUT_CONTROL.usa_TN_INPUT_CONTROL_DATA[11].in_Title_X_Offset := -27;
	Xus_TN_INPUT_CONTROL.usa_TN_INPUT_CONTROL_DATA[11].by_Title_Attr := BYTE#16#70;
	Xus_TN_INPUT_CONTROL.usa_TN_INPUT_CONTROL_DATA[11].st_Title_String := 'Telnet Interface        : <Enable >';

	Xus_TN_INPUT_CONTROL.usa_TN_INPUT_CONTROL_DATA[12].in_Type := INT#02;
	Xus_TN_INPUT_CONTROL.usa_TN_INPUT_CONTROL_DATA[12].in_Y := INT#18;
	Xus_TN_INPUT_CONTROL.usa_TN_INPUT_CONTROL_DATA[12].in_X := INT#44;
	Xus_TN_INPUT_CONTROL.usa_TN_INPUT_CONTROL_DATA[12].by_Attr_mF := BYTE#16#07;
	Xus_TN_INPUT_CONTROL.usa_TN_INPUT_CONTROL_DATA[12].by_Attr_oF := BYTE#16#70;
	Xus_TN_INPUT_CONTROL.usa_TN_INPUT_CONTROL_DATA[12].st_Input_Mask := '       ';
	Xus_TN_INPUT_CONTROL.usa_TN_INPUT_CONTROL_DATA[12].st_Input_Data := 'Enable#Disable';
	Xus_TN_INPUT_CONTROL.usa_TN_INPUT_CONTROL_DATA[12].st_Input_ToolTip := 'Push SPACE to Enable/Disable SNMP Interface (effective after reboot)';
	Xus_TN_INPUT_CONTROL.usa_TN_INPUT_CONTROL_DATA[12].in_Input_Option := INT#02;
	Xus_TN_INPUT_CONTROL.usa_TN_INPUT_CONTROL_DATA[12].in_Title_Y_Offset := INT#00;
	Xus_TN_INPUT_CONTROL.usa_TN_INPUT_CONTROL_DATA[12].in_Title_X_Offset := -27;
	Xus_TN_INPUT_CONTROL.usa_TN_INPUT_CONTROL_DATA[12].by_Title_Attr := BYTE#16#70;
	Xus_TN_INPUT_CONTROL.usa_TN_INPUT_CONTROL_DATA[12].st_Title_String := 'SNMP Interface          : <Enable >';

	Xus_TN_INPUT_CONTROL.usa_TN_INPUT_CONTROL_DATA[13].in_Type := INT#02;
	Xus_TN_INPUT_CONTROL.usa_TN_INPUT_CONTROL_DATA[13].in_Y := INT#20;
	Xus_TN_INPUT_CONTROL.usa_TN_INPUT_CONTROL_DATA[13].in_X := INT#44;
	Xus_TN_INPUT_CONTROL.usa_TN_INPUT_CONTROL_DATA[13].by_Attr_mF := BYTE#16#07;
	Xus_TN_INPUT_CONTROL.usa_TN_INPUT_CONTROL_DATA[13].by_Attr_oF := BYTE#16#70;
	Xus_TN_INPUT_CONTROL.usa_TN_INPUT_CONTROL_DATA[13].st_Input_Mask := '                                 ';
	Xus_TN_INPUT_CONTROL.usa_TN_INPUT_CONTROL_DATA[13].st_Input_Data := 'No reset#Reset Switch#Reset Switch to factory defaults';
	Xus_TN_INPUT_CONTROL.usa_TN_INPUT_CONTROL_DATA[13].st_Input_ToolTip := 'Push SPACE to select Reset Option';
	Xus_TN_INPUT_CONTROL.usa_TN_INPUT_CONTROL_DATA[13].in_Input_Option := INT#02;
	Xus_TN_INPUT_CONTROL.usa_TN_INPUT_CONTROL_DATA[13].in_Title_Y_Offset := INT#00;
	Xus_TN_INPUT_CONTROL.usa_TN_INPUT_CONTROL_DATA[13].in_Title_X_Offset := -27;
	Xus_TN_INPUT_CONTROL.usa_TN_INPUT_CONTROL_DATA[13].by_Title_Attr := BYTE#16#70;
	Xus_TN_INPUT_CONTROL.usa_TN_INPUT_CONTROL_DATA[13].st_Title_String := 'Reset                   : <No reset                         >';

	Xus_TN_INPUT_CONTROL.usa_TN_INPUT_CONTROL_DATA[14].in_Type := INT#02;
	Xus_TN_INPUT_CONTROL.usa_TN_INPUT_CONTROL_DATA[14].in_Y := INT#22;
	Xus_TN_INPUT_CONTROL.usa_TN_INPUT_CONTROL_DATA[14].in_X := INT#18;
	Xus_TN_INPUT_CONTROL.usa_TN_INPUT_CONTROL_DATA[14].by_Attr_mF := BYTE#16#07;
	Xus_TN_INPUT_CONTROL.usa_TN_INPUT_CONTROL_DATA[14].by_Attr_oF := BYTE#16#70;
	Xus_TN_INPUT_CONTROL.usa_TN_INPUT_CONTROL_DATA[14].st_Input_ToolTip := 'Apply and save ALL changes to permanent memory';
	Xus_TN_INPUT_CONTROL.usa_TN_INPUT_CONTROL_DATA[14].in_Input_Option := INT#01;
	Xus_TN_INPUT_CONTROL.usa_TN_INPUT_CONTROL_DATA[14].in_Title_Y_Offset := INT#00;
	Xus_TN_INPUT_CONTROL.usa_TN_INPUT_CONTROL_DATA[14].in_Title_X_Offset := INT#00;
	Xus_TN_INPUT_CONTROL.usa_TN_INPUT_CONTROL_DATA[14].by_Title_Attr := BYTE#16#70;
	Xus_TN_INPUT_CONTROL.usa_TN_INPUT_CONTROL_DATA[14].st_Title_String := '';
	Xus_TN_INPUT_CONTROL.usa_TN_INPUT_CONTROL_DATA[14].st_Input_Mask := '    ';
	Xus_TN_INPUT_CONTROL.usa_TN_INPUT_CONTROL_DATA[14].st_Input_Data := 'SAVE';

	Xus_TN_INPUT_CONTROL.usa_TN_INPUT_CONTROL_DATA[15].in_Type := INT#02;
	Xus_TN_INPUT_CONTROL.usa_TN_INPUT_CONTROL_DATA[15].in_Y := INT#22;
	Xus_TN_INPUT_CONTROL.usa_TN_INPUT_CONTROL_DATA[15].in_X := INT#11;
	Xus_TN_INPUT_CONTROL.usa_TN_INPUT_CONTROL_DATA[15].by_Attr_mF := BYTE#16#07;
	Xus_TN_INPUT_CONTROL.usa_TN_INPUT_CONTROL_DATA[15].by_Attr_oF := BYTE#16#70;
	Xus_TN_INPUT_CONTROL.usa_TN_INPUT_CONTROL_DATA[15].st_Input_ToolTip := 'Apply changes';
	Xus_TN_INPUT_CONTROL.usa_TN_INPUT_CONTROL_DATA[15].in_Input_Option := INT#01;
	Xus_TN_INPUT_CONTROL.usa_TN_INPUT_CONTROL_DATA[15].in_Title_Y_Offset := INT#00;
	Xus_TN_INPUT_CONTROL.usa_TN_INPUT_CONTROL_DATA[15].in_Title_X_Offset := INT#00;
	Xus_TN_INPUT_CONTROL.usa_TN_INPUT_CONTROL_DATA[15].by_Title_Attr := BYTE#16#70;
	Xus_TN_INPUT_CONTROL.usa_TN_INPUT_CONTROL_DATA[15].st_Title_String := '';
	Xus_TN_INPUT_CONTROL.usa_TN_INPUT_CONTROL_DATA[15].st_Input_Mask := '     ';
	Xus_TN_INPUT_CONTROL.usa_TN_INPUT_CONTROL_DATA[15].st_Input_Data := 'APPLY';

	Xus_TN_INPUT_CONTROL.usa_TN_INPUT_CONTROL_DATA[16].in_Type := INT#02;
	Xus_TN_INPUT_CONTROL.usa_TN_INPUT_CONTROL_DATA[16].in_Y := INT#22;
	Xus_TN_INPUT_CONTROL.usa_TN_INPUT_CONTROL_DATA[16].in_X := INT#03;
	Xus_TN_INPUT_CONTROL.usa_TN_INPUT_CONTROL_DATA[16].by_Attr_mF := BYTE#16#07;
	Xus_TN_INPUT_CONTROL.usa_TN_INPUT_CONTROL_DATA[16].by_Attr_oF := BYTE#16#70;
	Xus_TN_INPUT_CONTROL.usa_TN_INPUT_CONTROL_DATA[16].st_Input_ToolTip := 'Return to Main Menu';
	Xus_TN_INPUT_CONTROL.usa_TN_INPUT_CONTROL_DATA[16].in_Input_Option := INT#01;
	Xus_TN_INPUT_CONTROL.usa_TN_INPUT_CONTROL_DATA[16].in_Title_Y_Offset := INT#00;
	Xus_TN_INPUT_CONTROL.usa_TN_INPUT_CONTROL_DATA[16].in_Title_X_Offset := INT#00;
	Xus_TN_INPUT_CONTROL.usa_TN_INPUT_CONTROL_DATA[16].by_Title_Attr := BYTE#16#70;
	Xus_TN_INPUT_CONTROL.usa_TN_INPUT_CONTROL_DATA[16].st_Title_String := '';
	Xus_TN_INPUT_CONTROL.usa_TN_INPUT_CONTROL_DATA[16].st_Input_Mask := '      ';
	Xus_TN_INPUT_CONTROL.usa_TN_INPUT_CONTROL_DATA[16].st_Input_Data := 'LOGOUT';

	(* Control-Tool-Tip *)
	Xus_TN_INPUT_CONTROL.in_ToolTip_Y := INT#23;
	Xus_TN_INPUT_CONTROL.in_ToolTip_X := INT#00;
	Xus_TN_INPUT_CONTROL.by_ToolTip_Attr := BYTE#07;
	Xus_TN_INPUT_CONTROL.in_ToolTip_Size := INT#80;

	(* Control-Verwaltung initialisieren *)
	Xus_TN_INPUT_CONTROL.in_Count := INT#16;
	Xus_TN_INPUT_CONTROL.bo_Enable := TRUE;
	Xus_TN_INPUT_CONTROL.bo_Reset_Fokus := TRUE;

END_IF;

IF (Xus_TN_SCREEN.in_Page_Number = INT#05) THEN

	(* eingegebenen String übernehmen *)
	IF Xus_TN_INPUT_CONTROL.usa_TN_INPUT_CONTROL_DATA[16].bo_Input_Entered = TRUE THEN

		Xus_TN_INPUT_CONTROL.usa_TN_INPUT_CONTROL_DATA[16].bo_Input_Entered := FALSE;
		Xus_TN_SCREEN.in_Page_Number := INT#00;
	END_IF;
END_IF;

END_PROGRAM

// POUs/CONVERT/URL_DECODE
FUNCTION URL_DECODE : STRING(OSCAT_BASIC.STRING_LENGTH)
VAR_INPUT
	IN : STRING(OSCAT_BASIC.STRING_LENGTH);
END_VAR
VAR
	pos : INT;
	seq : STRING(3);
	new : STRING(1);
END_VAR


(*
version 1.2		10. may. 2010
programmer 	hugo
tested by		hugo

URL_DECODE checks a string if it contains non reserved characters represented by a % followed with the two digit hex code and converts them to their ascii code.
the non reserved characters are : [A..Z], [a..z], [0..9], -_.~
for example the character sequence '%23' will be converted to '#'.

*)

URL_DECODE := IN;
pos := FIND(URL_DECODE,'%');
WHILE pos > 0 DO
	seq := MID(URL_DECODE,2,pos + 1);
	new := OSCAT_BASIC.CHR_TO_STRING(DWORD_TO_BYTE(OSCAT_BASIC.HEX_TO_DWORD(seq)));
	URL_DECODE := REPLACE(URL_DECODE, new, 3, pos);
	pos := FIND(URL_DECODE,'%');
END_WHILE;


(* revision history
hm	27. apr. 2008	rev 1.0
	original version

hm	17. dec. 2008	rev 1.1
	changes name of function chr to chr_to_string

ks	10. mai. 2008	rev 1.2
	stringlength 250
*)

END_FUNCTION

// POUs/CONVERT/URL_ENCODE
FUNCTION URL_ENCODE : STRING(OSCAT_BASIC.STRING_LENGTH)
VAR_INPUT
	IN : STRING(OSCAT_BASIC.STRING_LENGTH);
END_VAR
VAR
	pt_in : POINTER TO ARRAY[1..255] OF BYTE;
	pt_out : POINTER TO ARRAY[1..256] OF BYTE;
	pos_in : INT;
	pos_out : INT;
	stop : INT;
	tb : BYTE;
END_VAR


(*
version 1.1		10. may. 2010
programmer 	hugo
tested by		hugo

URL_ENCODE checks a string if it contains only non reserved characters for an url.
the non reserved characters are : [A..Z], [a..z], [0..9], -_.~
if reserved characters are found then these characters are converted to %HH while HH is the Hexadezimal representation of the character in Alphabetic Letters.
for example the reserved character # will be converted to '%23'.

*)

pt_in  := ADR(in);
pt_out := ADR(URL_ENCODE);

(* scan the input string and convert unallowed characters *)
pos_in := 1;
stop := LEN(in);
FOR pos_out := 1 TO 250 DO
	IF pos_in > stop THEN
		EXIT;
	ELSIF IS_URLCHR(pt_in^[pos_in]) THEN
		pt_out^[pos_out] := pt_in^[pos_in];
		(* increment in by 1 *)
		pos_in := pos_in + 1;
	ELSE
		(* cannot fit 3 digits, exit *)
		IF pos_out > 248 THEN EXIT; END_IF;
		(* invalid character that needs to be converted *)
		pt_out^[pos_out] := 37;    (* start with % sign *)
		pos_out := pos_out + 1;
		(* need to add the two hex digits *)
		tb := SHR(pt_in^[pos_in],4);
		IF tb > 9 THEN
			pt_out^[pos_out] := tb + 55;
		ELSE
			pt_out^[pos_out] := tb + 48;
		END_IF;
		pos_out := pos_out + 1;
		tb := pt_in^[pos_in] AND 16#0F;
		IF tb > 9 THEN
			pt_out^[pos_out] := tb + 55;
		ELSE
			pt_out^[pos_out] := tb + 48;
		END_IF;
		(* increment in and out because out has to move 3 digits *)
		pos_in := pos_in + 1;
	END_IF;
END_FOR;

(* terminate the output string *)
pt_out^[pos_out] := 0;

(* revision history
hm	27. apr. 2008	rev 1.0
	original version

ks	10. mai. 2008	rev 1.1
	stringlength 250

*)

END_FUNCTION

// POUs/CONVERT/URL_TO_STRING
FUNCTION URL_TO_STRING : STRING(OSCAT_BASIC.STRING_LENGTH)
VAR_INPUT
	IN : URL;
END_VAR


(*
version 1.1		10. may. 2010
programmer 	hugo
tested by		oscat

URL_TO_STRING generates a string from URL information suppied in IN..

*)

(*

http://hans:geheim@www.example.org:80/demo/example.cgi?land=de&stadt=aa#abschnitt1
|         |         |                  |                                |   |                                    |                                    |
|         |         |                 Host                         |   Pfad                            Query                           Anker
|         |         Passwort                                  Port
|        Benutzer
Protokoll

*)

(* attach protocol *)
IF IN.PROTOCOL <> '' THEN URL_TO_STRING := CONCAT(IN.PROTOCOL,'://'); END_IF;

(* attach user and password *)
IF IN.USER <> '' THEN
	URL_TO_STRING := CONCAT(URL_TO_STRING, IN.USER);
	IF IN.PASSWORD <> '' THEN
		URL_TO_STRING := CONCAT(URL_TO_STRING, ':');
		URL_TO_STRING := CONCAT(URL_TO_STRING, IN.PASSWORD);
	END_IF;
	URL_TO_STRING := CONCAT(URL_TO_STRING, '@');
END_IF;

(* attach domain *)
URL_TO_STRING := CONCAT(URL_TO_STRING, IN.DOMAIN);

(* attach Port *)
IF IN.PORT > 0 THEN
	URL_TO_STRING := CONCAT(URL_TO_STRING, ':');
	URL_TO_STRING := CONCAT(URL_TO_STRING, WORD_TO_STRING(IN.PORT));
END_IF;

(* attach path *)
URL_TO_STRING := CONCAT(URL_TO_STRING, IN.PATH);

(* attach query *)
IF IN.QUERY <> '' THEN
	URL_TO_STRING := CONCAT(URL_TO_STRING, '?');
	URL_TO_STRING := CONCAT(URL_TO_STRING, IN.QUERY);
END_IF;

(* attach anchor *)
IF IN.ANCHOR <> '' THEN
	URL_TO_STRING := CONCAT(URL_TO_STRING, '#');
	URL_TO_STRING := CONCAT(URL_TO_STRING, IN.ANCHOR);
END_IF;

(* revision history
hm	18. apr 2008	rev 1.0
	original version

ks	10. mai. 2008	rev 1.1
	stringlength 250
*)

END_FUNCTION

// POUs/WEATHER/WORLD_WEATHER
FUNCTION_BLOCK WORLD_WEATHER
VAR_IN_OUT
	IP_C : IP_C; (* IP_Control Verwaltungsstruktur *)
	S_BUF : NETWORK_BUFFER;
	R_BUF : NETWORK_BUFFER;
	WW : WORLD_WEATHER_DATA;
END_VAR
VAR_INPUT
	ACTIVATE : BOOL;
	LATITUDE : REAL;
	LONGITUDE : REAL;
	KEY : STRING(30);
END_VAR
VAR_OUTPUT
	BUSY : BOOL;
	DONE : BOOL;
	ERROR_C : DWORD;
	ERROR_T : BYTE;
END_VAR
VAR
	URL_DATA : url;
	DNS_CLIENT : DNS_CLIENT;
	HTTP_GET : HTTP_GET;
	CPB : CSV_PARSER_BUF;
	last_state : BOOL;
	value_int : INT;
	value_real : REAL;
	v_real : REAL;
	state : INT;
	url_str : STRING(OSCAT_BASIC.STRING_LENGTH);
	offset : UDINT;
	size : INT;
	sep : BYTE;
	cnt : INT;
	day : INT;
	idx : INT;
	run : BYTE;
	result : BYTE;
	value : STRING(OSCAT_BASIC.STRING_LENGTH);
	pos : INT;
END_VAR

(*

version 1.5	11. may 2013
programmer 	ks
tested by	ks

WORLD_WEATHER lädt von worldweather.com eine Wetter csv-datei und analysiert die Daten und legt diese in einem Array ab
Die Wetterdaten werden für 5 tage aufbereitet

*)

CASE state OF

00:
	IF ACTIVATE AND NOT last_state THEN
		state := 20;
		DONE := FALSE;
		BUSY := TRUE;
		ERROR_C := DWORD#0;
		ERROR_T := BYTE#0;
	END_IF;

20: (* URL for DNS UND HTTP-GET *)
	(* Example: http://api.worldweatheronline.com/free/v1/weather.ashx?q=48.21,16.37&format=csv&num_of_days=5&key=xxxxxxxxxxxxxxxxxxxxxx *)
	url_str := CONCAT('http://api.worldweatheronline.com/free/v1/weather.ashx?q=',OSCAT_BASIC.REAL_TO_STRF(LATITUDE,6,D:='.'));
	url_str := CONCAT(url_str,',');
	url_str := CONCAT(url_str,OSCAT_BASIC.REAL_TO_STRF(LONGITUDE,6,D:='.'));
	url_str := CONCAT(url_str,'&format=csv&num_of_days=5&key=');
	url_str := CONCAT(url_str,key);

	URL_DATA:=STRING_TO_URL(STR:=url_str, DEFAULT_PROTOCOL:='', DEFAULT_PATH:='' );
	state := 40;

40:
	IF DNS_CLIENT.DONE THEN
		state := 60;
	ELSIF (DNS_CLIENT.ERROR > DWORD#00) THEN
		(* Fehlerbehandlung *)
		ERROR_C := DNS_CLIENT.ERROR;
	ERROR_T := BYTE#01;
		state   := 100;
	END_IF;

60:
	IF HTTP_GET.DONE THEN
		sep := 0;
		idx := 0;
		day := 0;
		cnt := 0;
		OFFSET := HTTP_GET.BODY_START; (* Start Offset vorgeben *)
		size := HTTP_GET.BODY_STOP; (* End Position *)
		run := 1; (* Element suchen *)
		state := 80;

	ELSIF (HTTP_GET.ERROR > DWORD#00) THEN
		(* Fehlerbehandlung *)
		ERROR_C := HTTP_GET.ERROR;
		ERROR_T := BYTE#02;
		state := 100;
	END_IF;

80:	IF run = 0 THEN (* kein Befehl mehr aktiv ? *)
		run := 1; (*  nächstes Element suchen  *)
		IF result = 1 OR result = 2 THEN
			value_int := 0;
			value_real := 0.0;
			(* automatische konvertierung in real und int ausführen *)
			IF LEN(value) <= 20 THEN
				v_real:=OSCAT_BASIC.FLOAT_TO_REAL(FLT:=value);
				IF OSCAT_BASIC.CHK_REAL(v_real) = 0 THEN (* !!! prüft auf gültigen REAL Wert, ansonsten stürzt Twincat ab !!!!  *)
					value_real := v_real;
					value_int := REAL_TO_INT(value_real);
				END_IF;
			END_IF;
			cnt := cnt + 1;


			IF cnt = 1 AND LEFT(value,1) <> '#' THEN
				cnt := 0;
			END_IF;

			IF cnt >=8 AND cnt <= 87 THEN
				IF cnt > 22 THEN
					CASE idx OF
					00:	WW.DAY[day].DATE_OF_DAY := value;
					01:	WW.DAY[day].TEMP_MAX_C := value_int;
					02:	WW.DAY[day].TEMP_MAX_F := value_int;
					03:	WW.DAY[day].TEMP_MIN_C := value_int;
					04:	WW.DAY[day].TEMP_MIN_F := value_int;
					05:	WW.DAY[day].WIND_SPEED_MILES := value_int;
					06:	WW.DAY[day].WIND_SPEED_KMPH := value_int;
					07:	WW.DAY[day].WIND_DIR_DEGREE := value_int;
					08:	WW.DAY[day].WIND_DIR16POINT := value;
					09:	WW.DAY[day].WEATHER_CODE := value_int;
					10:	pos := FIND(value, '/wsymbol_');
						WW.DAY[day].WEATHER_ICON := OSCAT_BASIC.DEC_TO_INT(MID(value,4,pos+9));
					11:	WW.DAY[day].WEATHER_DESC := value;
					12:	WW.DAY[day].PRECIPMM := value_real;
					END_CASE;
					idx := idx + 1;
					IF idx > 12 THEN
						idx := 0;
						day := day + 1;
					END_IF;
				ELSE
					CASE cnt OF
					08:	sep :=44; (* ab jetzt mit Trennzeichen arbeiten, *)
					09:	WW.CUR.OBSERVATION_TIME := value;
					10:	WW.CUR.TEMP_C := value_int;
					11:	WW.CUR.WEATHER_CODE := value_int;
					12:	pos := FIND(value, '/wsymbol_');
						WW.CUR.WEATHER_ICON := OSCAT_BASIC.DEC_TO_INT(MID(value,4,pos+9));
					13:	WW.CUR.WEATHER_DESC := value;
					14:	WW.CUR.WIND_SPEED_MILES := value_int;
					15:	WW.CUR.WIND_SPEED_KMPH := value_int;
					16:	WW.CUR.WIND_DIR_DEGREE := value_int;
					17:	WW.CUR.WIND_DIR16POINT := value;
					18:	WW.CUR.PRECIPMM := value_real;
					19:	WW.CUR.HUMIDITY := value_int;
					20:	WW.CUR.VISIBILITY := value_int;
					21:	WW.CUR.PRESSURE := value_int;
					22:	WW.CUR.CLOUDOVER := value_int;
					END_CASE;
				END_IF;
			END_IF;
		ELSIF result = 10 THEN (* nichts mehr gefunden *)
			DONE  := TRUE;
			run := 0; (* Auswertung beenden *)
			state := 100;
		END_IF;
	END_IF;

100:
	(* UNLOCK HTTP DATA *)
	IF (NOT HTTP_GET.DONE) THEN
		state := 0;
		BUSY := FALSE;
		DONE := ERROR_T = BYTE#0;
	END_IF;

END_CASE;

(* ---------------- DNS --------------- *)
DNS_CLIENT(	IP_C:=IP_C,
			S_BUF:=S_BUF,
			R_BUF:=R_BUF,
			DOMAIN:=URL_DATA.DOMAIN,
			IP4_DNS:=DWORD#00,
			ACTIVATE:=state=40 (* DNS Start *)
			);
(* nicht oder nicht direkt verwendete Parameter *)
(*	DWORD :=DNS_CLIENT.IP4;
	BOOL  :=DNS_CLIENT.DONE;
	BYTE  :=DNS_CLIENT.ERROR; *)
(* -------------------------------------*)

(* ------------- HTTP_GET --------------- *)
HTTP_GET(	IP_C:=IP_C,
			S_BUF:=S_BUF,
			R_BUF:=R_BUF,
			IP4:=DNS_CLIENT.IP4,
			GET:=state=60,
			MODE:=BYTE#2, (* HTTP 1.1 mit persistenter Verbindung *)
			UNLOCK_BUF:=state=100,
			URL_DATA:=URL_DATA
			);

(* nicht oder nicht direkt verwendete Parameter *)
(*	STRING := HTTP_GET.HTTP_STATUS;
	UINT :=HTTP_GET.HEADER_START;
	UINT :=HTTP_GET.HEADER_STOP;
	UINT :=HTTP_GET.BODY_START;
	UINT :=HTTP_GET.BODY_STOP;
	BOOL :=HTTP_GET.DONE;
	BYTE :=HTTP_GET.ERROR;
*)
(* -------------------------------------*)
CPB(SEP:=sep,RUN:=run,OFFSET:=OFFSET,VALUE:=value,PT:=R_BUF,RESULT=>result); (* CSV PARAMETER BUF *)

last_state := ACTIVATE;

(* revision history
ks	01.oct. 2010	rev 1.0
	original version

ks	01.feb. 2011	rev 1.1
	rücksetzen von cnt 

ks	07.apr. 2011	rev 1.2
	neue Domain "free.worldweatheronline.com" (Ab 30.04.2011 notwendig)

ks	05.jan. 2012	rev 1.3
	neues datenelement "icon" integriert, REAL_TO_STRF parameter D

ks	05.oct. 2012	rev 1.4
	workaround für chunked html data

ks	11.may. 2013	rev 1.5
	New worldwaether url and api key required (new API-Services)
*)

END_FUNCTION_BLOCK

// POUs/DEMO/WORLD_WEATHER_DEMO
PROGRAM WORLD_WEATHER_DEMO
VAR
	IP_C: IP_C;
	S_BUF: NETWORK_BUFFER;
	R_BUF: NETWORK_BUFFER;
	IP_CONTROL_1: IP_CONTROL;
	activate: BOOL := TRUE;
	done: BOOL;
	busy: BOOL;
	error_c: DWORD;
	error_t: BYTE;
	latitude: REAL := 48.21;
	longitude: REAL := 16.37;
	WORLD_WEATHER: WORLD_WEATHER;
	WW_DATA: WORLD_WEATHER_DATA;
	CLK_PRG: oscat_basic.CLK_PRG;
	WORLD_WEATHER_DESC_GE: WORLD_WEATHER_DESC_GE;
	WORLD_WEATHER_ICON_OSCAT: WORLD_WEATHER_ICON_OSCAT;
END_VAR
VAR // added by the converter: edge detectors and wires of the graphical bodies
    _w1 : ANY;
END_VAR

CLK_PRG(PT := t#3h); // oscat_basic.CLK_PRG
activate := CLK_PRG.Q;
WORLD_WEATHER(
    ACTIVATE := activate,
    LATITUDE := latitude,
    LONGITUDE := longitude,
    KEY := 'y94qq6e9dfk4ufwvv7eahnqs',
    IP_C := IP_C,
    S_BUF := S_BUF,
    R_BUF := R_BUF,
    WW := WW_DATA);
busy := WORLD_WEATHER.BUSY;
done := WORLD_WEATHER.DONE;
error_c := WORLD_WEATHER.ERROR_C;
error_t := WORLD_WEATHER.ERROR_T;
// Wetterbeschreibung auf Deutsch (optional)
WORLD_WEATHER_DESC_GE(ACTIVATE := done, WW := WW_DATA);
// ICONS nach OSCAT-Standard (optional)
WORLD_WEATHER_ICON_OSCAT(ACTIVATE := done, WW := WW_DATA);
// IP-Adresse des DNS-Server oder des DSL-Router
_w1 := oscat_basic.DWORD_OF_BYTE(B3 := 8, B2 := 8, B1 := 8, B0 := 8);
IP_CONTROL_1(IP := _w1, TIME_OUT := T#5s, IP_C := IP_C, S_BUF := S_BUF, R_BUF := R_BUF); // IP_CONTROL

END_PROGRAM

// POUs/WEATHER/WORLD_WEATHER_DESC_GE
FUNCTION_BLOCK WORLD_WEATHER_DESC_GE
VAR_IN_OUT
	WW : WORLD_WEATHER_DATA;
END_VAR
VAR_INPUT
	ACTIVATE : BOOL;
END_VAR
VAR
	act_last : BOOL;
	x : INT;
	y : INT;
	str : STRING(60);
	i : INT;
END_VAR

(*

version 1.0		04. may. 2011
programmer 		ks
tested by			ks

WORLD_WEATHER_DESC_GE ändert die englischen Wetterbeschreibungstexte auf deutsche Texte um
*)

IF ACTIVATE AND act_last = FALSE THEN
	i := 0;
	FOR y := 1 TO 12 DO
		CASE y OF
		1,3,5,7,9:		x :=  WW.DAY[i].WEATHER_CODE;
		2,4,6,8,10:	WW.DAY[i].WEATHER_DESC := str;
					i := i + 1;
		11:			x :=  WW.CUR.WEATHER_CODE;
		12:			WW.CUR.WEATHER_DESC := str;
		END_CASE;

		CASE x OF
			113	:	str := 'heiter/sonnig';
			116	:	str := 'stellenweise wolkig';
			119	:	str := 'wolkig';
			122	:	str := 'bewölkt';
			143	:	str := 'Nebel';
			176	:	str := 'stellenweise nahegelegener Regen';
			179	:	str := 'stellenweise nahegelegener Schneefall';
			182	:	str := 'stellenweise nahegelegener Eisregen';
			185	:	str := 'stellenweise gefrierender Niesel';
			200	:	str := 'nahegelegene Sturm';
			227	:	str := 'Schneetreiben';
			230	:	str := 'Schneesturm';
			248	:	str := 'Nebel';
			260	:	str := 'gefrierender Nebel';
			263	:	str := 'stellenweise leichter Nieselregen';
			266	:	str := 'leichter Niesel';
			281	:	str := 'gefrierender Nieselregen';
			284	:	str := 'stark gefrierender Nieselregen';
			293	:	str := 'stellenweise leichter Regen';
			296	:	str := 'leichter Regen';
			299	:	str := 'zeitweise etwas Regen';
			302	:	str := 'mäßiger Regen';
			305	:	str := 'zeitweise etwas starker Regen';
			308	:	str := 'starker Regen';
			311	:	str := 'leichter gefrierender Regen';
			314	:	str := 'mäßiger oder starker Eisregen';
			317	:	str := 'leichter Eisregen';
			320	:	str := 'mäßiger oder starker Eisregen';
			323	:	str := 'stellenweise leichter Schneefall';
			326	:	str := 'leichter Scheefall';
			329	:	str := 'stellenweise moderater Schneefall';
			332	:	str := 'mäßiger Schnee';
			335	:	str := 'stellenweise starker Scheefall';
			338	:	str := 'starker Schneefall';
			350	:	str := 'Hagel';
			353	:	str := 'leichte Regenfälle';
			356	:	str := 'mäßiger oder starker Regenfall';
			359	:	str := 'sintflutartige Regenfälle';
			362	:	str := 'leichter Eisregen';
			365	:	str := 'mäßiger oder starker Eisregen';
			368	:	str := 'leichte Schneeschauer';
			371	:	str := 'mäßiger oder starker Schneefall';
			374	:	str := 'leichter Hagel';
			377	:	str := 'mäßiger oder starker Hagel';
			386	:	str := 'stellenweise leichter Regen in Gewittergebiet';
			389	:	str := 'mäßiger oder starker Regen in Gewittergebiet';
			392	:	str := 'stellenweise leichter Schneefall in Gewittergebiet';
			395	:	str := 'mäßiger oder starker Schnee in Gewittergebiet';
		ELSE
			str := 	'nicht verfügbar';
		END_CASE;
	END_FOR;
END_IF;
act_last := ACTIVATE;

(* revision history
ks	04. may. 2011	rev 1.0
	original version
*)

END_FUNCTION_BLOCK

// POUs/WEATHER/WORLD_WEATHER_ICON_OSCAT
FUNCTION_BLOCK WORLD_WEATHER_ICON_OSCAT
VAR_IN_OUT
	WW : WORLD_WEATHER_DATA;
END_VAR
VAR_INPUT
	ACTIVATE : BOOL;
END_VAR
VAR
	dat : ARRAY[0..41] OF INT := [0,14,12,9,9,0,7,7,0,2,2,3,3,1,0,0,17,4,4,3,3,1,0,0,17,2,2,3,3,1,0,0,17,2,4,3,3,1,0,0,17,0];
	act_last : BOOL;
	x : INT;
	i : INT;
END_VAR

(*

version 1.0		04. may. 2011
programmer 		ks
tested by			ks

WORLD_WEATHER_ICON_OSCAT ändert die ICON Nummer auf den OSCAT-Standard um
*)

IF ACTIVATE AND act_last = FALSE THEN
	x := LIMIT(0,WW.CUR.WEATHER_ICON,41);
	WW.CUR.WEATHER_ICON := dat[x];
	FOR i := 0 TO 4 DO
		x := LIMIT(0,WW.DAY[i].WEATHER_ICON,41);
		WW.DAY[i].WEATHER_ICON := dat[x];
	END_FOR;
END_IF;
act_last := ACTIVATE;

(* revision history
ks	04. may. 2011	rev 1.0
	original version
*)

END_FUNCTION_BLOCK

// POUs/DEMO/YAHOO_WEATHER_DEMO
PROGRAM YAHOO_WEATHER_DEMO
VAR
	IP_C: IP_C;
	S_BUF: NETWORK_BUFFER;
	R_BUF: NETWORK_BUFFER;
	IP_CONTROL_1: IP_CONTROL;
	activate: BOOL;
	done: BOOL;
	busy: BOOL;
	error_c: DWORD;
	error_t: BYTE;
	YAHOO_WEATHER: YAHOO_WEATHER;
	YW_DATA: YAHOO_WEATHER_DATA;
	CLK_PRG: oscat_basic.CLK_PRG;
	YAHOO_WEATHER_DESC_GE: YAHOO_WEATHER_DESC_GE;
	YAHOO_WEATHER_ICON_OSCAT: YAHOO_WEATHER_ICON_OSCAT;
END_VAR
VAR // added by the converter: edge detectors and wires of the graphical bodies
    _w1 : ANY;
END_VAR

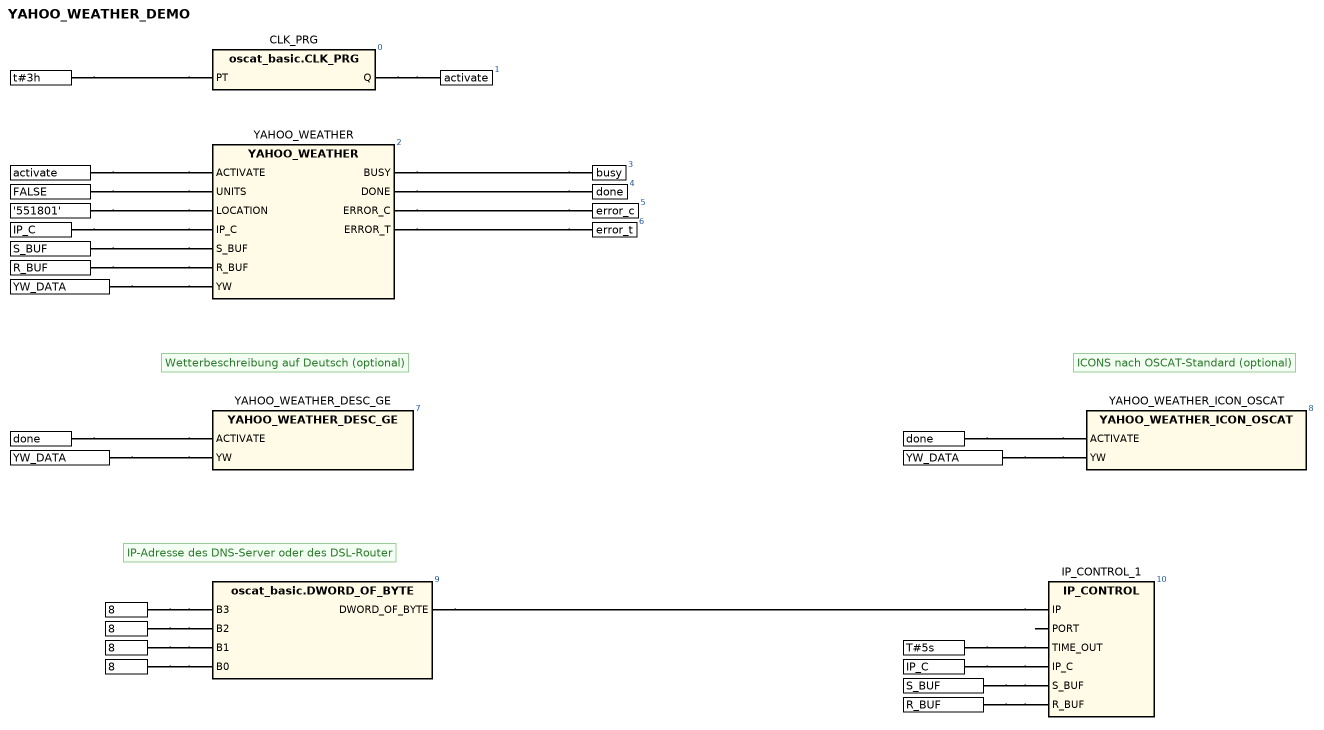
CLK_PRG(PT := t#3h); // oscat_basic.CLK_PRG
activate := CLK_PRG.Q;
YAHOO_WEATHER(
    ACTIVATE := activate,
    UNITS := FALSE,
    LOCATION := '551801',
    IP_C := IP_C,
    S_BUF := S_BUF,
    R_BUF := R_BUF,
    YW := YW_DATA);
busy := YAHOO_WEATHER.BUSY;
done := YAHOO_WEATHER.DONE;
error_c := YAHOO_WEATHER.ERROR_C;
error_t := YAHOO_WEATHER.ERROR_T;
// Wetterbeschreibung auf Deutsch (optional)
YAHOO_WEATHER_DESC_GE(ACTIVATE := done, YW := YW_DATA);
// ICONS nach OSCAT-Standard (optional)
YAHOO_WEATHER_ICON_OSCAT(ACTIVATE := done, YW := YW_DATA);
// IP-Adresse des DNS-Server oder des DSL-Router
_w1 := oscat_basic.DWORD_OF_BYTE(B3 := 8, B2 := 8, B1 := 8, B0 := 8);
IP_CONTROL_1(IP := _w1, TIME_OUT := T#5s, IP_C := IP_C, S_BUF := S_BUF, R_BUF := R_BUF); // IP_CONTROL

END_PROGRAM

// POUs/WEATHER/YAHOO_WEATHER_DESC_GE
FUNCTION_BLOCK YAHOO_WEATHER_DESC_GE
VAR_IN_OUT
	YW : YAHOO_WEATHER_DATA;
END_VAR
VAR_INPUT
	ACTIVATE : BOOL;
END_VAR
VAR
	act_last : BOOL;
	x : INT;
	y : INT;
	str : STRING(40);
END_VAR

(*
version 1.1		01. jun. 2016
programmer 		ks
tested by			ks

YAHOO_WEATHER_DESC_GE ändert die englischen Wetterbeschreibungstexte auf deutsche Texte um
*)

IF ACTIVATE AND act_last = FALSE THEN
	FOR y := 1 TO 12 DO
		CASE y OF
		01:	x := YW.CUR_CONDITIONS_CODE;

		02:	YW.CUR_CONDITIONS_TEXT := str;
			x := YW.FORECAST_TODAY_CODE;
		03:	YW.FORECAST_TODAY_TEXT := str;
			x := YW.FORECAST_DAY[1].CODE;
		04:	YW.FORECAST_DAY[1].TEXT := str;
			x := YW.FORECAST_DAY[2].CODE;
		05:	YW.FORECAST_DAY[2].TEXT := str;
			x := YW.FORECAST_DAY[3].CODE;
		06:	YW.FORECAST_DAY[3].TEXT := str;
			x := YW.FORECAST_DAY[4].CODE;
		07:	YW.FORECAST_DAY[4].TEXT := str;
			x := YW.FORECAST_DAY[5].CODE;
		08:	YW.FORECAST_DAY[5].TEXT := str;
			x := YW.FORECAST_DAY[6].CODE;
		09:	YW.FORECAST_DAY[6].TEXT := str;
			x := YW.FORECAST_DAY[7].CODE;
		10:	YW.FORECAST_DAY[7].TEXT := str;
			x := YW.FORECAST_DAY[8].CODE;
		11:	YW.FORECAST_DAY[8].TEXT := str;
			x := YW.FORECAST_DAY[9].CODE;
		12:	YW.FORECAST_DAY[9].TEXT := str;
		END_CASE;

		CASE x OF
		00:	str := 'Wirbelsturm';
		01:	str := 'Tropensturm';
		02:	str := 'Wirbelsturm';
		03:	str := 'starkes Gewitter ';
		04:	str := 'Gewitter';
		05:	str := 'Schneeregen';
		06:	str := 'Schneeregen';
		07:	str := 'Schneeregen';
		08:	str := 'gefrierender Nieselregen';
		09:	str := 'Nieselregen';
		10:	str := 'gefrierender Regen';
		11:	str := 'Regenfälle';
		12:	str := 'Regenfälle';
		13:	str := 'Schneegestöber';
		14:	str := 'leichte Schneefälle';
		15:	str := 'Schneetreiben';
		16:	str := 'Schnee';
		17:	str := 'Hagel';
		18:	str := 'Schneeregen';
		19:	str := 'Staub';
		20:	str := 'nebelig';
		21:	str := 'Dunst';
		22:	str := 'rauchig';
		23:	str := 'stürmisch';
		24:	str := 'windig';
		25:	str := 'kalt';
		26:	str := 'bewölkt';
		27:	str := 'meist bewölkt';
		28:	str := 'meist bewölkt';
		29:	str := 'teilweise bewölkt';
		30:	str := 'teilweise bewölkt';
		31:	str := 'klar';
		32:	str := 'sonnig';
		33:	str := 'heiter';
		34:	str := 'heiter';
		35:	str := 'Regen und Hagel';
		36:	str := 'heiß';
		37:	str := 'örtliche Gewitter';
		38:	str := 'vereinzelte Gewitter';
		39:	str := 'vereinzelte Gewitter';
		40:	str := 'vereinzelte Regenfälle';
		41:	str := 'schwere Schneefälle';
		42:	str := 'vereinzelte Schneefälle';
		43:	str := 'schwere Schneefälle';
		44:	str := 'teilweise bewölkt';
		45:	str := 'gewittrige Regenfälle';
		46:	str := 'Schneefälle';
		47:	str := 'örtliche gewittrige Regenfälle';
		ELSE
			str := 'nicht verfügbar';
		END_CASE;
	END_FOR;
END_IF;
act_last := ACTIVATE;

(* revision history
ks	04. may. 2011	rev 1.0
	original version
ks	01. jun. 2016	rev 1.1
	komplette überarbeitung auf neue yahoo-api

*)

END_FUNCTION_BLOCK

// POUs/WEATHER/YAHOO_WEATHER_ICON_OSCAT
FUNCTION_BLOCK YAHOO_WEATHER_ICON_OSCAT
VAR_IN_OUT
	YW : YAHOO_WEATHER_DATA;
END_VAR
VAR_INPUT
	ACTIVATE : BOOL;
END_VAR
VAR
	dat : ARRAY[0..48] OF INT := [4,2,2,4,17,1,3,1,2,2,2,2,2,3,3,3,3,5,3,6,7,14,8,9,9,10,9,11,12,11,12,13,14,15,16,4,14,4,17,2,2,3,3,3,12,2,3,4,0];
	act_last : BOOL;
	x : INT;
	idx : INT;
END_VAR

(*
version 1.1		01. jun. 2016
programmer 		ks
tested by			ks

YAHOO_WEATHER_ICON_OSCAT ändert die ICON Nummer auf den OSCAT-Standard um
*)

IF ACTIVATE AND act_last = FALSE THEN
	x := MIN(YW.CUR_CONDITIONS_CODE,48);
	YW.CUR_CONDITIONS_ICON := dat[x];
	x := MIN(YW.FORECAST_TODAY_CODE,48);
	YW.FORECAST_TODAY_ICON := dat[x];
	FOR idx := 1 TO 9 DO
		x := MIN(YW.FORECAST_DAY[idx].CODE,48);
		YW.FORECAST_DAY[idx].ICON := dat[x];
	END_FOR;
END_IF;
act_last := ACTIVATE;

(* revision history
ks	04. may. 2011	rev 1.0
	original version

ks	01. jun. 2016	rev 1.1
	komplette überarbeitung auf neue yahoo-api
*)

END_FUNCTION_BLOCK
